FUNCTION_BLOCK RunSignal Extends CommonBase
VAR_INPUT
END_VAR
VAR_OUTPUT
	raw : BOOL;
	debouncedOn : BOOL;
	debouncedOff : BOOL;
END_VAR
VAR
	input AT%I* : BOOL;
END_VAR
VAR PERSISTENT
	debouncedOnTimer : TON;
	debouncedOffTimer : TOn;
END_VAR


raw := input;

debouncedOnTimer(IN:= input, PT:= , Q=> debouncedOn, ET=> );
debouncedOffTimer(IN:= NOT input, PT:= , Q=> debouncedoff, ET=> );

METHOD ConfigureRead : CellDataBlock
VAR_INPUT
	mode : eModes;
END_VAR
ConfigureRead.signal.widthOn := TO_WORD(debouncedOnTimer.PT);
ConfigureRead.signal.widthOff := TO_WORD(debouncedOffTimer.PT);
END_METHOD

METHOD ConfigureWrite : BOOL
VAR_INPUT
	input : CellDataBlock;
	mode : eModes;
END_VAR
debouncedOffTimer.PT := TO_TIME(input.signal.widthOff);
debouncedOnTimer.PT := TO_TIME(input.signal.widthOn);
END_METHOD

METHOD FB_init : BOOL
VAR_INPUT
	bInitRetains : BOOL; // if TRUE, the retain variables are initialized (warm start / cold start)
	bInCopyCode : BOOL;  // if TRUE, the instance afterwards gets moved into the copy code (online change)
END_VAR
IF bInitRetains THEN
	debouncedOnTimer.PT := T#100MS;
	debouncedOffTimer.PT := T#100ms;
END_IF
END_METHOD

METHOD Monitor : CellDataBlock
VAR_INPUT
END_VAR
VAR CONSTANT
	indexDebouncedOn : INT := 0;
	indexDebouncedOff : INT := 1;
	indexRaw : INT := 2;
END_VAR
Monitor.signal.widthOffCount := TO_WORD(debouncedOffTimer.ET);
Monitor.signal.widthOnCount := TO_WORD(debouncedOnTimer.ET);

Monitor.signal.outputWord.indexDebouncedOn := debouncedOn;
Monitor.signal.outputWord.indexDebouncedOff := debouncedOff;
Monitor.signal.outputWord.indexRaw := raw;
END_METHOD

END_FUNCTION_BLOCK

(* stored: Version 1.1.0.1, ProductVersion 3.1.4022.10
   POU RunSignal: Id {2f1f5cd2-5e24-47f9-8ea9-a8607aa3166e}, SpecialFunc None
   Folder CommonBase: Id {ffc1ce20-d0f1-44f8-8792-2f966b14be1c}
   Method ConfigureRead: Id {a12d05cb-7391-4f12-9f9c-52f812ce9a7d}
   Method ConfigureWrite: Id {6bdc42d6-cbc4-4a8a-bfcd-b648766e27b5}
   Method FB_init: Id {87ea7c0f-d400-4141-b585-3dd2db5cdf88}
   Method Monitor: Id {502646b2-e6fc-4522-882f-20960251e59a} *)
